FUNCTION F_DeviceTwin_GetPublisherTopic : STRING
VAR_INPUT
END_VAR
VAR
END_VAR

F_DeviceTwin_GetPublisherTopic := '$$iothub/twin/PATCH/properties/reported/?$rid=42';

END_FUNCTION

(* stored: Version 1.1.0.1, ProductVersion 3.1.4022.3
   POU F_DeviceTwin_GetPublisherTopic: Id {733722ae-9871-4e2e-887b-1f0a4ad18904}, SpecialFunc None *)
